FUNCTION_BLOCK AxisCommand IMPLEMENTS itfAxisCommand
VAR_INPUT
	_done			: REFERENCE TO BOOL;
	_busy			: REFERENCE TO BOOL;
	_active			: REFERENCE TO BOOL;
	_commandAborted	: REFERENCE TO BOOL;
	_error			: REFERENCE TO BOOL;
	_errorId		: REFERENCE TO UDINT;
END_VAR

{warning 'Add method implementation '}
METHOD Abort : UDINT
END_METHOD

PROPERTY Active : BOOL
GET
Active := _active;
END_GET
END_PROPERTY

PROPERTY Busy : BOOL
GET
Busy := _busy;
END_GET
END_PROPERTY

{warning 'Add property implementation'}
PROPERTY Command : MC_COMMAND_REF
GET
END_GET
END_PROPERTY

PROPERTY CommandAborted : BOOL
GET
CommandAborted := _commandAborted;
END_GET
END_PROPERTY

PROPERTY Done : BOOL
GET
Done := done;
END_GET
END_PROPERTY

PROPERTY Error : BOOL
GET
Error := _error;
END_GET
END_PROPERTY

PROPERTY ErrorId : UDINT
GET
ErrorId := _errorId;
END_GET
END_PROPERTY

{warning 'Add method implementation '}
METHOD Update		: UDINT
VAR_INPUT
	Position		: REAL;
	Velocity		: REAL;
	EndVelocity		: REAL;
	Acceleration	: REAL;
	Deceleration	: REAL;
	Jerk			: REAL;
END_VAR
END_METHOD

{warning 'Add method implementation '}
METHOD Wait			: UDINT (* This method only makes sense in the IEC 61499 environment*)
VAR_INPUT
	Timeout			: TIME;
	AbortOnTimeout	: BOOL;
END_VAR
END_METHOD

END_FUNCTION_BLOCK

(* stored: Version 1.1.0.1, ProductVersion 3.1.4024.12
   POU AxisCommand: Id {c76c5803-28be-4710-93f6-5a71bd9fc9ca}, SpecialFunc None
   Method Abort: Id {eeb96b01-61d8-4b66-b3ec-f32db0335b5a}
   Property Active: Id {fe0aef6d-bfb5-4e5f-864b-673d26bc6b15}
   Get Get: Id {b05b3318-e0fc-46ae-b5e0-1a660d87afe5}
   Property Busy: Id {5dfcac70-a4d5-41e5-abc5-ea54ee828e11}
   Get Get: Id {f9b30e7c-13a3-419e-b39c-68a13f0fb48b}
   Property Command: Id {d61d00e8-3411-4d8e-bb8b-b2b5d34ff95e}
   Get Get: Id {ad98bdab-7e15-466c-b6ef-5872a58211ad}
   Property CommandAborted: Id {24438402-1760-4305-84f6-06e65cd9fc74}
   Get Get: Id {02663dbc-db4c-40b0-bade-bd39632d1d3d}
   Property Done: Id {897fee26-f9c5-4bee-b06c-28626cc7c2b8}
   Get Get: Id {37d79d3e-9829-46c3-869c-ecfb60318c14}
   Property Error: Id {10a2d898-cfee-46dc-bd2e-cdc969fa1c4e}
   Get Get: Id {f0a68396-dcfc-4d53-9c62-0da3adf60e9b}
   Property ErrorId: Id {cf43a610-f12e-47a5-acbb-5d66995282b2}
   Get Get: Id {c64fb9ff-8bcc-42ee-b026-f3362a78a7d5}
   Method Update: Id {c2f5fcf0-750d-4b1c-9388-a34979dddc0e}
   Method Wait: Id {0957b123-f5bf-4c00-ae39-c97b3c60159b} *)
